FUNCTION_BLOCK FB_RecipeAnalogControlInputSequencer
VAR_INPUT
	rampTime: UINT;
END_VAR
VAR_IN_OUT
	rRecipe: ARRAY[1..(GVL_CONSTANT.NumAnalogController)] OF REAL;
END_VAR
VAR
	i: INT;
END_VAR

FOR i:= 1 TO E_aAnalogInputIO_Index.E_PV_EPC_04 DO
	IF 0.0 < GVL_IO.aMaxValueController[i] THEN
		GVL_IO.aController[i].input.restart := TRUE;
		GVL_IO.aController[i].input.rampTime := rampTime; 
		GVL_IO.aController[i].input.targetValue := rRecipe[i] / GVL_IO.aMaxValueController[i] * GVL_CONSTANT.EL3064MaxValueH;
	END_IF
END_FOR

FOR i:= E_aAnalogInputIO_Index.E_PV_Susceptor_Temp TO E_aAnalogInputIO_Index.E_PV_susceptorRotation DO
	GVL_IO.aController[i].input.restart := TRUE;
	GVL_IO.aController[i].input.rampTime := rampTime;
	GVL_IO.aController[i].input.targetValue := rRecipe[i];
END_FOR

END_FUNCTION_BLOCK

(* stored: Version 1.1.0.1, ProductVersion 3.1.4026.11
   POU FB_RecipeAnalogControlInputSequencer: Id {baa4a425-4968-4360-81b7-f83562b782ba}, SpecialFunc None *)
